NA													:=			0    		,
Standby                                             :=          1           ,
IOLP                                                :=          2           ,
PNB                                                 :=          3           ,
TBOT                                                :=          4           ,
LP_VISIONSHUTTLE_L                                  :=          1500        ,
LP_VISIONSHUTTLE_R                                  :=          1600        ,
LP_LE                                               :=          1900        ,
LP_L01                                              :=          1901        ,
LP_L02                                              :=          1902        ,
LP_RE                                               :=          1903        ,
LP_R01                                              :=          1904        ,
LP_R02                                              :=          1905        ,
LP_L                                                :=          1910        ,
LP_R                                                :=          1911        ,
LP_LE_STACKER_01                                    :=          2000        ,
LP_LE_STACKER_01_LIFT                               :=          2001        ,
LP_LE_STACKER_01_STOPPER_01                         :=          2002        ,
LP_LE_STACKER_01_STOPPER_02                         :=          2003        ,
LP_LE_STACKER_02                                    :=          2050        ,
LP_LE_STACKER_02_LIFT                               :=          2051        ,
LP_LE_STACKER_02_STOPPER_01                         :=          2052        ,
LP_LE_STACKER_02_STOPPER_02                         :=          2053        ,
LP_LE_CONVEYOR                                      :=          2200        ,
LP_LE_CONVEYOR_STACKER_01_PRE                       :=          2250        ,
LP_LE_CONVEYOR_STACKER_01                           :=          2251        ,
LP_LE_CONVEYOR_STACKER_01_POST                      :=          2252        ,
LP_LE_CONVEYOR_STACKER_02                           :=          2300        ,
LP_L01_STACKER_01                                   :=          3000        ,
LP_L01_STACKER_01_LIFT                              :=          3001        ,
LP_L01_STACKER_01_STOPPER_01                        :=          3002        ,
LP_L01_STACKER_01_STOPPER_02                        :=          3003        ,
LP_L01_STACKER_02                                   :=          3050        ,
LP_L01_STACKER_02_LIFT                              :=          3051        ,
LP_L01_STACKER_02_STOPPER_01                        :=          3052        ,
LP_L01_STACKER_02_STOPPER_02                        :=          3053        ,
LP_L01_CONVEYOR_01                                  :=          3110        ,
LP_L01_CONVEYOR_02                                  :=          3120        ,
LP_L01_CONVEYOR_STACKER_01_PRE                      :=          3125        ,
LP_L01_CONVEYOR_STACKER_01                          :=          3126        ,
LP_L01_CONVEYOR_STACKER_01_POST                     :=          3127        ,
LP_L01_CONVEYOR_STACKER_02                          :=          3128        ,
LP_L01_CONVEYOR_STACKER_02_POST                     :=          3129        ,
LP_L01_EPORT                                        :=          3130        ,
LP_L01_EPORT_STANDBY                                :=          3131        ,
LP_L01_EPORT_STOPPER_01                             :=          3132        ,
LP_L01_EPORT_STOPPER_02                             :=          3133        ,
LP_L01_VISION                                       :=          3140        ,
LP_L01_UPORT                                        :=          3151        ,
LP_L02_STACKER_01                                   :=          3200        ,
LP_L02_STACKER_01_LIFT                              :=          3201        ,
LP_L02_STACKER_01_STOPPER_01                        :=          3202        ,
LP_L02_STACKER_01_STOPPER_02                        :=          3203        ,
LP_L02_STACKER_02                                   :=          3250        ,
LP_L02_STACKER_02_LIFT                              :=          3251        ,
LP_L02_STACKER_02_STOPPER_01                        :=          3252        ,
LP_L02_STACKER_02_STOPPER_02                        :=          3253        ,
LP_L02_CONVEYOR_01                                  :=          3310        ,
LP_L02_CONVEYOR_02                                  :=          3320        ,
LP_L02_CONVEYOR_STACKER_01_PRE                      :=          3325        ,
LP_L02_CONVEYOR_STACKER_01                          :=          3326        ,
LP_L02_CONVEYOR_STACKER_01_POST                     :=          3327        ,
LP_L02_CONVEYOR_STACKER_02                          :=          3328        ,
LP_L02_CONVEYOR_STACKER_02_POST                     :=          3329        ,
LP_L02_EPORT                                        :=          3330        ,
LP_L02_EPORT_STANDBY                                :=          3331        ,
LP_L02_EPORT_STOPPER_01                             :=          3332        ,
LP_L02_EPORT_STOPPER_02                             :=          3333        ,
LP_L02_VISION                                       :=          3340        ,
LP_L02_UPORT                                        :=          3351        ,
LP_RE_STACKER_01                                    :=          4000        ,
LP_RE_STACKER_01_LIFT                               :=          4001        ,
LP_RE_STACKER_01_STOPPER_01                         :=          4002        ,
LP_RE_STACKER_01_STOPPER_02                         :=          4003        ,
LP_RE_STACKER_02                                    :=          4050        ,
LP_RE_STACKER_02_LIFT                               :=          4051        ,
LP_RE_STACKER_02_STOPPER_01                         :=          4052        ,
LP_RE_STACKER_02_STOPPER_02                         :=          4053        ,
LP_RE_CONVEYOR                                      :=          4200        ,
LP_RE_CONVEYOR_STACKER_01_PRE                       :=          4250        ,
LP_RE_CONVEYOR_STACKER_01                           :=          4251        ,
LP_RE_CONVEYOR_STACKER_01_POST                      :=          4252        ,
LP_RE_CONVEYOR_STACKER_02                           :=          4300        ,
LP_R01_STACKER_01                                   :=          5000        ,
LP_R01_STACKER_01_LIFT                              :=          5001        ,
LP_R01_STACKER_01_STOPPER_01                        :=          5002        ,
LP_R01_STACKER_01_STOPPER_02                        :=          5003        ,
LP_R01_STACKER_02                                   :=          5050        ,
LP_R01_STACKER_02_LIFT                              :=          5051        ,
LP_R01_STACKER_02_STOPPER_01                        :=          5052        ,
LP_R01_STACKER_02_STOPPER_02                        :=          5053        ,
LP_R01_CONVEYOR_01                                  :=          5110        ,
LP_R01_CONVEYOR_02                                  :=          5120        ,
LP_R01_CONVEYOR_STACKER_01_PRE                      :=          5125        ,
LP_R01_CONVEYOR_STACKER_01                          :=          5126        ,
LP_R01_CONVEYOR_STACKER_01_POST                     :=          5127        ,
LP_R01_CONVEYOR_STACKER_02                          :=          5128        ,
LP_R01_CONVEYOR_STACKER_02_POST                     :=          5129        ,
LP_R01_EPORT                                        :=          5130        ,
LP_R01_EPORT_STANDBY                                :=          5131        ,
LP_R01_EPORT_STOPPER_01                             :=          5132        ,
LP_R01_EPORT_STOPPER_02                             :=          5133        ,
LP_R01_VISION                                       :=          5140        ,
LP_R01_UPORT                                        :=          5151        ,
LP_R02_STACKER_01                                   :=          5200        ,
LP_R02_STACKER_01_LIFT                              :=          5201        ,
LP_R02_STACKER_01_STOPPER_01                        :=          5202        ,
LP_R02_STACKER_01_STOPPER_02                        :=          5203        ,
LP_R02_STACKER_02                                   :=          5250        ,
LP_R02_STACKER_02_LIFT                              :=          5251        ,
LP_R02_STACKER_02_STOPPER_01                        :=          5252        ,
LP_R02_STACKER_02_STOPPER_02                        :=          5253        ,
LP_R02_CONVEYOR_01                                  :=          5310        ,
LP_R02_CONVEYOR_02                                  :=          5320        ,
LP_R02_CONVEYOR_STACKER_01_PRE                      :=          5325        ,
LP_R02_CONVEYOR_STACKER_01                          :=          5326        ,
LP_R02_CONVEYOR_STACKER_01_POST                     :=          5327        ,
LP_R02_CONVEYOR_STACKER_02                          :=          5328        ,
LP_R02_CONVEYOR_STACKER_02_POST                     :=          5329        ,
LP_R02_EPORT                                        :=          5330        ,
LP_R02_EPORT_STANDBY                                :=          5331        ,
LP_R02_EPORT_STOPPER_01                             :=          5332        ,
LP_R02_EPORT_STOPPER_02                             :=          5333        ,
LP_R02_VISION                                       :=          5340        ,
LP_R02_UPORT                                        :=          5351        ,
TTS                                                 :=          10000       ,
TTS_SHUTTLE_01                                      :=          10100       ,
TTS_SHUTTLE_01_SERVICE                              :=          10101       ,
TTS_SHUTTLE_01_PARK                                 :=          10102       ,
TTS_SHUTTLE_01_CONVEYOR                             :=          10103       ,
TTS_SHUTTLE_02                                      :=          10200       ,
TTS_SHUTTLE_02_SERVICE                              :=          10201       ,
TTS_SHUTTLE_02_CONVEYOR                             :=          10202       ,
TTS_SHUTTLE_03                                      :=          10300       ,
TTS_SHUTTLE_03_SERVICE                              :=          10301       ,
TTS_SHUTTLE_03_PARK                                 :=          10302       ,
TTS_SHUTTLE_03_CONVEYOR                             :=          10303       ,
PNB_DOOR_TOP_LEFT                                   :=          20001       ,
PNB_DOOR_TOP_RIGHT                                  :=          20002       ,
PNB_DOOR_BOTTOM                                     :=          20003       ,
PNB_LANE_01                                         :=          21000       ,
PNB_LANE_01_CONVEYOR                                :=          21001       ,
PNB_LANE_02                                         :=          21050       ,
PNB_LANE_02_CONVEYOR                                :=          21051       ,
PNB_LANE_03                                         :=          21150       ,
PNB_LANE_03_CONVEYOR                                :=          21151       ,
PNB_LANE_04                                         :=          21200       ,
PNB_LANE_04_CONVEYOR                                :=          21201       ,
PNB_LANE_05                                         :=          21350       ,
PNB_LANE_05_CONVEYOR                                :=          21351       ,
PNB_LANE_06                                         :=          21400       ,
PNB_LANE_06_CONVEYOR                                :=          21401       ,
PNB_LANE_07                                         :=          21450       ,
PNB_LANE_07_CONVEYOR                                :=          21451       ,
PNB_LANE_08                                         :=          21500       ,
PNB_LANE_08_CONVEYOR                                :=          21501       ,
PNB_GANTRY_01                                       :=          22500       ,
PNB_GANTRY_01_PARK                                  :=          22501       ,
PNB_UPCAM_L                                         :=          22502       ,
PNB_RFID_L                                          :=          22503       ,
PNB_RFID_L_01                                       :=          22504       ,
PNB_RFID_L_02                                       :=          22505       ,
PNB_GANTRY_01_SERVICE                               :=          22506       ,
PNB_GANTRY_01_HEAD_A01                              :=          22550       ,
PNB_GANTRY_01_HEAD_A02                              :=          22560       ,
PNB_GANTRY_01_HEAD_A03                              :=          22570       ,
PNB_GANTRY_01_HEAD_A04                              :=          22580       ,
PNB_GANTRY_02                                       :=          23000       ,
PNB_GANTRY_02_PARK                                  :=          23001       ,
PNB_UPCAM_R                                         :=          23002       ,
PNB_RFID_R                                          :=          23003       ,
PNB_RFID_R_01                                       :=          23004       ,
PNB_RFID_R_02                                       :=          23005       ,
PNB_GANTRY_02_SERVICE                               :=          23006       ,
PNB_GANTRY_02_HEAD_A01                              :=          23050       ,
PNB_GANTRY_02_HEAD_A02                              :=          23060       ,
PNB_GANTRY_02_HEAD_A03                              :=          23070       ,
PNB_GANTRY_02_HEAD_A04                              :=          23080       ,
PRECISOR_UL                                         :=          24000       ,
PRECISOR_UL_CLEAN                                   :=          24001       ,
PRECISOR_UL_01                                      :=          24002       ,
PRECISOR_UL_02                                      :=          24003       ,
PRECISOR_UL_CLEAN_READID                            :=          24004       ,
PRECISOR_UL_01_READID                               :=          24005       ,
PRECISOR_UL_02_READID                               :=          24006       ,
PRECISOR_UL_A01_01                                  :=          24011       ,
PRECISOR_UL_A01_02                                  :=          24012       ,
PRECISOR_UL_A02_01                                  :=          24021       ,
PRECISOR_UL_A02_02                                  :=          24022       ,
PRECISOR_UL_A03_01                                  :=          24031       ,
PRECISOR_UL_A03_02                                  :=          24032       ,
PRECISOR_UL_A04_01                                  :=          24041       ,
PRECISOR_UL_A04_02                                  :=          24042       ,
PRECISOR_UL_B01_01                                  :=          24061       ,
PRECISOR_UL_B01_02                                  :=          24062       ,
PRECISOR_UL_B02_01                                  :=          24071       ,
PRECISOR_UL_B02_02                                  :=          24072       ,
PRECISOR_UL_B03_01                                  :=          24081       ,
PRECISOR_UL_B03_02                                  :=          24082       ,
PRECISOR_UL_B04_01                                  :=          24091       ,
PRECISOR_UL_B04_02                                  :=          24092       ,
PRECISOR_UL_C01_01                                  :=          24111       ,
PRECISOR_UL_C01_02                                  :=          24112       ,
PRECISOR_UL_C02_01                                  :=          24121       ,
PRECISOR_UL_C02_02                                  :=          24122       ,
PRECISOR_UL_C03_01                                  :=          24131       ,
PRECISOR_UL_C03_02                                  :=          24132       ,
PRECISOR_UL_C04_01                                  :=          24141       ,
PRECISOR_UL_C04_02                                  :=          24142       ,
PRECISOR_UL_D01_01                                  :=          24161       ,
PRECISOR_UL_D01_02                                  :=          24162       ,
PRECISOR_UL_D02_01                                  :=          24171       ,
PRECISOR_UL_D02_02                                  :=          24172       ,
PRECISOR_UL_D03_01                                  :=          24181       ,
PRECISOR_UL_D03_02                                  :=          24182       ,
PRECISOR_UL_D04_01                                  :=          24191       ,
PRECISOR_UL_D04_02                                  :=          24192       ,
PRECISOR_UR                                         :=          24500       ,
PRECISOR_UR_CLEAN                                   :=          24501       ,
PRECISOR_UR_01                                      :=          24502       ,
PRECISOR_UR_02                                      :=          24503       ,
PRECISOR_UR_CLEAN_READID                            :=          24504       ,
PRECISOR_UR_01_READID                               :=          24505       ,
PRECISOR_UR_02_READID                               :=          24506       ,
PRECISOR_UR_A01_01                                  :=          24511       ,
PRECISOR_UR_A01_02                                  :=          24512       ,
PRECISOR_UR_A02_01                                  :=          24521       ,
PRECISOR_UR_A02_02                                  :=          24522       ,
PRECISOR_UR_A03_01                                  :=          24531       ,
PRECISOR_UR_A03_02                                  :=          24532       ,
PRECISOR_UR_A04_01                                  :=          24541       ,
PRECISOR_UR_A04_02                                  :=          24542       ,
PRECISOR_UR_B01_01                                  :=          24561       ,
PRECISOR_UR_B01_02                                  :=          24562       ,
PRECISOR_UR_B02_01                                  :=          24571       ,
PRECISOR_UR_B02_02                                  :=          24572       ,
PRECISOR_UR_B03_01                                  :=          24581       ,
PRECISOR_UR_B03_02                                  :=          24582       ,
PRECISOR_UR_B04_01                                  :=          24591       ,
PRECISOR_UR_B04_02                                  :=          24592       ,
PRECISOR_UR_C01_01                                  :=          24611       ,
PRECISOR_UR_C01_02                                  :=          24612       ,
PRECISOR_UR_C02_01                                  :=          24621       ,
PRECISOR_UR_C02_02                                  :=          24622       ,
PRECISOR_UR_C03_01                                  :=          24631       ,
PRECISOR_UR_C03_02                                  :=          24632       ,
PRECISOR_UR_C04_01                                  :=          24641       ,
PRECISOR_UR_C04_02                                  :=          24642       ,
PRECISOR_UR_D01_01                                  :=          24661       ,
PRECISOR_UR_D01_02                                  :=          24662       ,
PRECISOR_UR_D02_01                                  :=          24671       ,
PRECISOR_UR_D02_02                                  :=          24672       ,
PRECISOR_UR_D03_01                                  :=          24681       ,
PRECISOR_UR_D03_02                                  :=          24682       ,
PRECISOR_UR_D04_01                                  :=          24691       ,
PRECISOR_UR_D04_02                                  :=          24692       ,
PRECISOR_DL                                         :=          25000       ,
PRECISOR_DL_CLEAN                                   :=          25001       ,
PRECISOR_DL_01                                      :=          25002       ,
PRECISOR_DL_02                                      :=          25003       ,
PRECISOR_DL_CLEAN_READID                            :=          25004       ,
PRECISOR_DL_01_READID                               :=          25005       ,
PRECISOR_DL_02_READID                               :=          25006       ,
PRECISOR_DL_A01_01                                  :=          25011       ,
PRECISOR_DL_A01_02                                  :=          25012       ,
PRECISOR_DL_A02_01                                  :=          25021       ,
PRECISOR_DL_A02_02                                  :=          25022       ,
PRECISOR_DL_A03_01                                  :=          25031       ,
PRECISOR_DL_A03_02                                  :=          25032       ,
PRECISOR_DL_A04_01                                  :=          25041       ,
PRECISOR_DL_A04_02                                  :=          25042       ,
PRECISOR_DL_B01_01                                  :=          25061       ,
PRECISOR_DL_B01_02                                  :=          25062       ,
PRECISOR_DL_B02_01                                  :=          25071       ,
PRECISOR_DL_B02_02                                  :=          25072       ,
PRECISOR_DL_B03_01                                  :=          25081       ,
PRECISOR_DL_B03_02                                  :=          25082       ,
PRECISOR_DL_B04_01                                  :=          25091       ,
PRECISOR_DL_B04_02                                  :=          25092       ,
PRECISOR_DL_C01_01                                  :=          25111       ,
PRECISOR_DL_C01_02                                  :=          25112       ,
PRECISOR_DL_C02_01                                  :=          25121       ,
PRECISOR_DL_C02_02                                  :=          25122       ,
PRECISOR_DL_C03_01                                  :=          25131       ,
PRECISOR_DL_C03_02                                  :=          25132       ,
PRECISOR_DL_C04_01                                  :=          25141       ,
PRECISOR_DL_C04_02                                  :=          25142       ,
PRECISOR_DL_D01_01                                  :=          25161       ,
PRECISOR_DL_D01_02                                  :=          25162       ,
PRECISOR_DL_D02_01                                  :=          25171       ,
PRECISOR_DL_D02_02                                  :=          25172       ,
PRECISOR_DL_D03_01                                  :=          25181       ,
PRECISOR_DL_D03_02                                  :=          25182       ,
PRECISOR_DL_D04_01                                  :=          25191       ,
PRECISOR_DL_D04_02                                  :=          25192       ,
PRECISOR_DR                                         :=          25500       ,
PRECISOR_DR_CLEAN                                   :=          25501       ,
PRECISOR_DR_01                                      :=          25502       ,
PRECISOR_DR_02                                      :=          25503       ,
PRECISOR_DR_CLEAN_READID                            :=          25504       ,
PRECISOR_DR_01_READID                               :=          25505       ,
PRECISOR_DR_02_READID                               :=          25506       ,
PRECISOR_DR_A01_01                                  :=          25511       ,
PRECISOR_DR_A01_02                                  :=          25512       ,
PRECISOR_DR_A02_01                                  :=          25521       ,
PRECISOR_DR_A02_02                                  :=          25522       ,
PRECISOR_DR_A03_01                                  :=          25531       ,
PRECISOR_DR_A03_02                                  :=          25532       ,
PRECISOR_DR_A04_01                                  :=          25541       ,
PRECISOR_DR_A04_02                                  :=          25542       ,
PRECISOR_DR_B01_01                                  :=          25561       ,
PRECISOR_DR_B01_02                                  :=          25562       ,
PRECISOR_DR_B02_01                                  :=          25571       ,
PRECISOR_DR_B02_02                                  :=          25572       ,
PRECISOR_DR_B03_01                                  :=          25581       ,
PRECISOR_DR_B03_02                                  :=          25582       ,
PRECISOR_DR_B04_01                                  :=          25591       ,
PRECISOR_DR_B04_02                                  :=          25592       ,
PRECISOR_DR_C01_01                                  :=          25611       ,
PRECISOR_DR_C01_02                                  :=          25612       ,
PRECISOR_DR_C02_01                                  :=          25621       ,
PRECISOR_DR_C02_02                                  :=          25622       ,
PRECISOR_DR_C03_01                                  :=          25631       ,
PRECISOR_DR_C03_02                                  :=          25632       ,
PRECISOR_DR_C04_01                                  :=          25641       ,
PRECISOR_DR_C04_02                                  :=          25642       ,
PRECISOR_DR_D01_01                                  :=          25661       ,
PRECISOR_DR_D01_02                                  :=          25662       ,
PRECISOR_DR_D02_01                                  :=          25671       ,
PRECISOR_DR_D02_02                                  :=          25672       ,
PRECISOR_DR_D03_01                                  :=          25681       ,
PRECISOR_DR_D03_02                                  :=          25682       ,
PRECISOR_DR_D04_01                                  :=          25691       ,
PRECISOR_DR_D04_02                                  :=          25692       ,
TBOT_L                                              :=          30000       ,
TBOT_L_RFID                                         :=          30001       ,
TBOT_L_SERVICE                                      :=          30002       ,
TBOT_L_PARK                                         :=          30003       ,
TBOT_L_HEAD_A01                                     :=          30020       ,
TBOT_L_HEAD_A02                                     :=          30040       ,
TBOT_L_HEAD_A03                                     :=          30060       ,
TBOT_L_HEAD_A04                                     :=          30080       ,
TBOT_L_HEAD_B01                                     :=          30100       ,
TBOT_L_HEAD_B02                                     :=          30120       ,
TBOT_L_HEAD_B03                                     :=          30140       ,
TBOT_L_HEAD_B04                                     :=          30160       ,
TBOT_L_HEAD_C01                                     :=          30180       ,
TBOT_L_HEAD_C02                                     :=          30200       ,
TBOT_L_HEAD_C03                                     :=          30220       ,
TBOT_L_HEAD_C04                                     :=          30240       ,
TBOT_L_HEAD_D01                                     :=          30260       ,
TBOT_L_HEAD_D02                                     :=          30280       ,
TBOT_L_HEAD_D03                                     :=          30300       ,
TBOT_L_HEAD_D04                                     :=          30320       ,
TBOT_R                                              :=          30500       ,
TBOT_R_RFID                                         :=          30501       ,
TBOT_R_SERVICE                                      :=          30502       ,
TBOT_R_PARK                                         :=          30503       ,
TBOT_R_HEAD_A01                                     :=          30520       ,
TBOT_R_HEAD_A02                                     :=          30540       ,
TBOT_R_HEAD_A03                                     :=          30560       ,
TBOT_R_HEAD_A04                                     :=          30580       ,
TBOT_R_HEAD_B01                                     :=          30600       ,
TBOT_R_HEAD_B02                                     :=          30620       ,
TBOT_R_HEAD_B03                                     :=          30640       ,
TBOT_R_HEAD_B04                                     :=          30660       ,
TBOT_R_HEAD_C01                                     :=          30680       ,
TBOT_R_HEAD_C02                                     :=          30700       ,
TBOT_R_HEAD_C03                                     :=          30720       ,
TBOT_R_HEAD_C04                                     :=          30740       ,
TBOT_R_HEAD_D01                                     :=          30760       ,
TBOT_R_HEAD_D02                                     :=          30780       ,
TBOT_R_HEAD_D03                                     :=          30800       ,
TBOT_R_HEAD_D04                                     :=          30820       ,
COLUMN_LA                                           :=          35000       ,
COLUMN_LB                                           :=          35100       ,
COLUMN_LC                                           :=          35200       ,
COLUMN_RA                                           :=          35300       ,
COLUMN_RB                                           :=          35400       ,
COLUMN_RC                                           :=          35500       ,
LEVEL_LA01                                          :=          36000       ,
LEVEL_LA02                                          :=          36010       ,
LEVEL_LA03                                          :=          36020       ,
LEVEL_LA04                                          :=          36030       ,
LEVEL_LA05                                          :=          36040       ,
LEVEL_LA06                                          :=          36050       ,
LEVEL_LB01                                          :=          36060       ,
LEVEL_LB02                                          :=          36070       ,
LEVEL_LB03                                          :=          36080       ,
LEVEL_LB04                                          :=          36090       ,
LEVEL_LB05                                          :=          36100       ,
LEVEL_LB06                                          :=          36110       ,
LEVEL_LC01                                          :=          36120       ,
LEVEL_LC02                                          :=          36130       ,
LEVEL_LC03                                          :=          36140       ,
LEVEL_LC04                                          :=          36150       ,
LEVEL_LC05                                          :=          36160       ,
LEVEL_LC06                                          :=          36170       ,
LEVEL_RA01                                          :=          37000       ,
LEVEL_RA02                                          :=          37010       ,
LEVEL_RA03                                          :=          37020       ,
LEVEL_RA04                                          :=          37030       ,
LEVEL_RA05                                          :=          37040       ,
LEVEL_RA06                                          :=          37050       ,
LEVEL_RB01                                          :=          37060       ,
LEVEL_RB02                                          :=          37070       ,
LEVEL_RB03                                          :=          37080       ,
LEVEL_RB04                                          :=          37090       ,
LEVEL_RB05                                          :=          37100       ,
LEVEL_RB06                                          :=          37110       ,
LEVEL_RC01                                          :=          37120       ,
LEVEL_RC02                                          :=          37130       ,
LEVEL_RC03                                          :=          37140       ,
LEVEL_RC04                                          :=          37150       ,
LEVEL_RC05                                          :=          37160       ,
LEVEL_RC06                                          :=          37170       ,
CELL_LA101_TESTER                                   :=          45000       ,
CELL_LA101_TESTER_SOCKET_A01                        :=          45001       ,
CELL_LA101_TESTER_SOCKET_A02                        :=          45002       ,
CELL_LA101_TESTER_SOCKET_A03                        :=          45003       ,
CELL_LA101_TESTER_SOCKET_A04                        :=          45004       ,
CELL_LA101_TESTER_SOCKET_B01                        :=          45011       ,
CELL_LA101_TESTER_SOCKET_B02                        :=          45012       ,
CELL_LA101_TESTER_SOCKET_B03                        :=          45013       ,
CELL_LA101_TESTER_SOCKET_B04                        :=          45014       ,
CELL_LA101_TESTER_SOCKET_C01                        :=          45021       ,
CELL_LA101_TESTER_SOCKET_C02                        :=          45022       ,
CELL_LA101_TESTER_SOCKET_C03                        :=          45023       ,
CELL_LA101_TESTER_SOCKET_C04                        :=          45024       ,
CELL_LA101_TESTER_SOCKET_D01                        :=          45031       ,
CELL_LA101_TESTER_SOCKET_D02                        :=          45032       ,
CELL_LA101_TESTER_SOCKET_D03                        :=          45033       ,
CELL_LA101_TESTER_SOCKET_D04                        :=          45034       ,
CELL_LA101_TESTER_FRONT                             :=          45035       ,
CELL_LA101_AP                                       :=          45050       ,
CELL_LA101_AP_TH_A01                                :=          45051       ,
CELL_LA101_AP_TH_A02                                :=          45052       ,
CELL_LA101_AP_TH_A03                                :=          45053       ,
CELL_LA101_AP_TH_A04                                :=          45054       ,
CELL_LA101_AP_TH_B01                                :=          45061       ,
CELL_LA101_AP_TH_B02                                :=          45062       ,
CELL_LA101_AP_TH_B03                                :=          45063       ,
CELL_LA101_AP_TH_B04                                :=          45064       ,
CELL_LA101_AP_TH_C01                                :=          45071       ,
CELL_LA101_AP_TH_C02                                :=          45072       ,
CELL_LA101_AP_TH_C03                                :=          45073       ,
CELL_LA101_AP_TH_C04                                :=          45074       ,
CELL_LA101_AP_TH_D01                                :=          45081       ,
CELL_LA101_AP_TH_D02                                :=          45082       ,
CELL_LA101_AP_TH_D03                                :=          45083       ,
CELL_LA101_AP_TH_D04                                :=          45084       ,
CELL_LA201_TESTER                                   :=          45100       ,
CELL_LA201_TESTER_SOCKET_A01                        :=          45101       ,
CELL_LA201_TESTER_SOCKET_A02                        :=          45102       ,
CELL_LA201_TESTER_SOCKET_A03                        :=          45103       ,
CELL_LA201_TESTER_SOCKET_A04                        :=          45104       ,
CELL_LA201_TESTER_SOCKET_B01                        :=          45111       ,
CELL_LA201_TESTER_SOCKET_B02                        :=          45112       ,
CELL_LA201_TESTER_SOCKET_B03                        :=          45113       ,
CELL_LA201_TESTER_SOCKET_B04                        :=          45114       ,
CELL_LA201_TESTER_SOCKET_C01                        :=          45121       ,
CELL_LA201_TESTER_SOCKET_C02                        :=          45122       ,
CELL_LA201_TESTER_SOCKET_C03                        :=          45123       ,
CELL_LA201_TESTER_SOCKET_C04                        :=          45124       ,
CELL_LA201_TESTER_SOCKET_D01                        :=          45131       ,
CELL_LA201_TESTER_SOCKET_D02                        :=          45132       ,
CELL_LA201_TESTER_SOCKET_D03                        :=          45133       ,
CELL_LA201_TESTER_SOCKET_D04                        :=          45134       ,
CELL_LA201_TESTER_FRONT                             :=          45135       ,
CELL_LA201_AP                                       :=          45150       ,
CELL_LA201_AP_TH_A01                                :=          45151       ,
CELL_LA201_AP_TH_A02                                :=          45152       ,
CELL_LA201_AP_TH_A03                                :=          45153       ,
CELL_LA201_AP_TH_A04                                :=          45154       ,
CELL_LA201_AP_TH_B01                                :=          45161       ,
CELL_LA201_AP_TH_B02                                :=          45162       ,
CELL_LA201_AP_TH_B03                                :=          45163       ,
CELL_LA201_AP_TH_B04                                :=          45164       ,
CELL_LA201_AP_TH_C01                                :=          45171       ,
CELL_LA201_AP_TH_C02                                :=          45172       ,
CELL_LA201_AP_TH_C03                                :=          45173       ,
CELL_LA201_AP_TH_C04                                :=          45174       ,
CELL_LA201_AP_TH_D01                                :=          45181       ,
CELL_LA201_AP_TH_D02                                :=          45182       ,
CELL_LA201_AP_TH_D03                                :=          45183       ,
CELL_LA201_AP_TH_D04                                :=          45184       ,
CELL_LA301_TESTER                                   :=          45200       ,
CELL_LA301_TESTER_SOCKET_A01                        :=          45201       ,
CELL_LA301_TESTER_SOCKET_A02                        :=          45202       ,
CELL_LA301_TESTER_SOCKET_A03                        :=          45203       ,
CELL_LA301_TESTER_SOCKET_A04                        :=          45204       ,
CELL_LA301_TESTER_SOCKET_B01                        :=          45211       ,
CELL_LA301_TESTER_SOCKET_B02                        :=          45212       ,
CELL_LA301_TESTER_SOCKET_B03                        :=          45213       ,
CELL_LA301_TESTER_SOCKET_B04                        :=          45214       ,
CELL_LA301_TESTER_SOCKET_C01                        :=          45221       ,
CELL_LA301_TESTER_SOCKET_C02                        :=          45222       ,
CELL_LA301_TESTER_SOCKET_C03                        :=          45223       ,
CELL_LA301_TESTER_SOCKET_C04                        :=          45224       ,
CELL_LA301_TESTER_SOCKET_D01                        :=          45231       ,
CELL_LA301_TESTER_SOCKET_D02                        :=          45232       ,
CELL_LA301_TESTER_SOCKET_D03                        :=          45233       ,
CELL_LA301_TESTER_SOCKET_D04                        :=          45234       ,
CELL_LA301_AP                                       :=          45250       ,
CELL_LA301_AP_TH_A01                                :=          45251       ,
CELL_LA301_AP_TH_A02                                :=          45252       ,
CELL_LA301_AP_TH_A03                                :=          45253       ,
CELL_LA301_AP_TH_A04                                :=          45254       ,
CELL_LA301_AP_TH_B01                                :=          45261       ,
CELL_LA301_AP_TH_B02                                :=          45262       ,
CELL_LA301_AP_TH_B03                                :=          45263       ,
CELL_LA301_AP_TH_B04                                :=          45264       ,
CELL_LA301_AP_TH_C01                                :=          45271       ,
CELL_LA301_AP_TH_C02                                :=          45272       ,
CELL_LA301_AP_TH_C03                                :=          45273       ,
CELL_LA301_AP_TH_C04                                :=          45274       ,
CELL_LA301_AP_TH_D01                                :=          45281       ,
CELL_LA301_AP_TH_D02                                :=          45282       ,
CELL_LA301_AP_TH_D03                                :=          45283       ,
CELL_LA301_AP_TH_D04                                :=          45284       ,
CELL_LA401_TESTER                                   :=          45300       ,
CELL_LA401_TESTER_SOCKET_A01                        :=          45301       ,
CELL_LA401_TESTER_SOCKET_A02                        :=          45302       ,
CELL_LA401_TESTER_SOCKET_A03                        :=          45303       ,
CELL_LA401_TESTER_SOCKET_A04                        :=          45304       ,
CELL_LA401_TESTER_SOCKET_B01                        :=          45311       ,
CELL_LA401_TESTER_SOCKET_B02                        :=          45312       ,
CELL_LA401_TESTER_SOCKET_B03                        :=          45313       ,
CELL_LA401_TESTER_SOCKET_B04                        :=          45314       ,
CELL_LA401_TESTER_SOCKET_C01                        :=          45321       ,
CELL_LA401_TESTER_SOCKET_C02                        :=          45322       ,
CELL_LA401_TESTER_SOCKET_C03                        :=          45323       ,
CELL_LA401_TESTER_SOCKET_C04                        :=          45324       ,
CELL_LA401_TESTER_SOCKET_D01                        :=          45331       ,
CELL_LA401_TESTER_SOCKET_D02                        :=          45332       ,
CELL_LA401_TESTER_SOCKET_D03                        :=          45333       ,
CELL_LA401_TESTER_SOCKET_D04                        :=          45334       ,
CELL_LA401_AP                                       :=          45350       ,
CELL_LA401_AP_TH_A01                                :=          45351       ,
CELL_LA401_AP_TH_A02                                :=          45352       ,
CELL_LA401_AP_TH_A03                                :=          45353       ,
CELL_LA401_AP_TH_A04                                :=          45354       ,
CELL_LA401_AP_TH_B01                                :=          45361       ,
CELL_LA401_AP_TH_B02                                :=          45362       ,
CELL_LA401_AP_TH_B03                                :=          45363       ,
CELL_LA401_AP_TH_B04                                :=          45364       ,
CELL_LA401_AP_TH_C01                                :=          45371       ,
CELL_LA401_AP_TH_C02                                :=          45372       ,
CELL_LA401_AP_TH_C03                                :=          45373       ,
CELL_LA401_AP_TH_C04                                :=          45374       ,
CELL_LA401_AP_TH_D01                                :=          45381       ,
CELL_LA401_AP_TH_D02                                :=          45382       ,
CELL_LA401_AP_TH_D03                                :=          45383       ,
CELL_LA401_AP_TH_D04                                :=          45384       ,
CELL_LA501_TESTER                                   :=          45400       ,
CELL_LA501_TESTER_SOCKET_A01                        :=          45401       ,
CELL_LA501_TESTER_SOCKET_A02                        :=          45402       ,
CELL_LA501_TESTER_SOCKET_A03                        :=          45403       ,
CELL_LA501_TESTER_SOCKET_A04                        :=          45404       ,
CELL_LA501_TESTER_SOCKET_B01                        :=          45411       ,
CELL_LA501_TESTER_SOCKET_B02                        :=          45412       ,
CELL_LA501_TESTER_SOCKET_B03                        :=          45413       ,
CELL_LA501_TESTER_SOCKET_B04                        :=          45414       ,
CELL_LA501_TESTER_SOCKET_C01                        :=          45421       ,
CELL_LA501_TESTER_SOCKET_C02                        :=          45422       ,
CELL_LA501_TESTER_SOCKET_C03                        :=          45423       ,
CELL_LA501_TESTER_SOCKET_C04                        :=          45424       ,
CELL_LA501_TESTER_SOCKET_D01                        :=          45431       ,
CELL_LA501_TESTER_SOCKET_D02                        :=          45432       ,
CELL_LA501_TESTER_SOCKET_D03                        :=          45433       ,
CELL_LA501_TESTER_SOCKET_D04                        :=          45434       ,
CELL_LA501_AP                                       :=          45450       ,
CELL_LA501_AP_TH_A01                                :=          45451       ,
CELL_LA501_AP_TH_A02                                :=          45452       ,
CELL_LA501_AP_TH_A03                                :=          45453       ,
CELL_LA501_AP_TH_A04                                :=          45454       ,
CELL_LA501_AP_TH_B01                                :=          45461       ,
CELL_LA501_AP_TH_B02                                :=          45462       ,
CELL_LA501_AP_TH_B03                                :=          45463       ,
CELL_LA501_AP_TH_B04                                :=          45464       ,
CELL_LA501_AP_TH_C01                                :=          45471       ,
CELL_LA501_AP_TH_C02                                :=          45472       ,
CELL_LA501_AP_TH_C03                                :=          45473       ,
CELL_LA501_AP_TH_C04                                :=          45474       ,
CELL_LA501_AP_TH_D01                                :=          45481       ,
CELL_LA501_AP_TH_D02                                :=          45482       ,
CELL_LA501_AP_TH_D03                                :=          45483       ,
CELL_LA501_AP_TH_D04                                :=          45484       ,
CELL_LA601_TESTER                                   :=          45500       ,
CELL_LA601_TESTER_SOCKET_A01                        :=          45501       ,
CELL_LA601_TESTER_SOCKET_A02                        :=          45502       ,
CELL_LA601_TESTER_SOCKET_A03                        :=          45503       ,
CELL_LA601_TESTER_SOCKET_A04                        :=          45504       ,
CELL_LA601_TESTER_SOCKET_B01                        :=          45511       ,
CELL_LA601_TESTER_SOCKET_B02                        :=          45512       ,
CELL_LA601_TESTER_SOCKET_B03                        :=          45513       ,
CELL_LA601_TESTER_SOCKET_B04                        :=          45514       ,
CELL_LA601_TESTER_SOCKET_C01                        :=          45521       ,
CELL_LA601_TESTER_SOCKET_C02                        :=          45522       ,
CELL_LA601_TESTER_SOCKET_C03                        :=          45523       ,
CELL_LA601_TESTER_SOCKET_C04                        :=          45524       ,
CELL_LA601_TESTER_SOCKET_D01                        :=          45531       ,
CELL_LA601_TESTER_SOCKET_D02                        :=          45532       ,
CELL_LA601_TESTER_SOCKET_D03                        :=          45533       ,
CELL_LA601_TESTER_SOCKET_D04                        :=          45534       ,
CELL_LA601_AP                                       :=          45550       ,
CELL_LA601_AP_TH_A01                                :=          45551       ,
CELL_LA601_AP_TH_A02                                :=          45552       ,
CELL_LA601_AP_TH_A03                                :=          45553       ,
CELL_LA601_AP_TH_A04                                :=          45554       ,
CELL_LA601_AP_TH_B01                                :=          45561       ,
CELL_LA601_AP_TH_B02                                :=          45562       ,
CELL_LA601_AP_TH_B03                                :=          45563       ,
CELL_LA601_AP_TH_B04                                :=          45564       ,
CELL_LA601_AP_TH_C01                                :=          45571       ,
CELL_LA601_AP_TH_C02                                :=          45572       ,
CELL_LA601_AP_TH_C03                                :=          45573       ,
CELL_LA601_AP_TH_C04                                :=          45574       ,
CELL_LA601_AP_TH_D01                                :=          45581       ,
CELL_LA601_AP_TH_D02                                :=          45582       ,
CELL_LA601_AP_TH_D03                                :=          45583       ,
CELL_LA601_AP_TH_D04                                :=          45584       ,
CELL_LB101_TESTER                                   :=          46000       ,
CELL_LB101_TESTER_SOCKET_A01                        :=          46001       ,
CELL_LB101_TESTER_SOCKET_A02                        :=          46002       ,
CELL_LB101_TESTER_SOCKET_A03                        :=          46003       ,
CELL_LB101_TESTER_SOCKET_A04                        :=          46004       ,
CELL_LB101_TESTER_SOCKET_B01                        :=          46011       ,
CELL_LB101_TESTER_SOCKET_B02                        :=          46012       ,
CELL_LB101_TESTER_SOCKET_B03                        :=          46013       ,
CELL_LB101_TESTER_SOCKET_B04                        :=          46014       ,
CELL_LB101_TESTER_SOCKET_C01                        :=          46021       ,
CELL_LB101_TESTER_SOCKET_C02                        :=          46022       ,
CELL_LB101_TESTER_SOCKET_C03                        :=          46023       ,
CELL_LB101_TESTER_SOCKET_C04                        :=          46024       ,
CELL_LB101_TESTER_SOCKET_D01                        :=          46031       ,
CELL_LB101_TESTER_SOCKET_D02                        :=          46032       ,
CELL_LB101_TESTER_SOCKET_D03                        :=          46033       ,
CELL_LB101_TESTER_SOCKET_D04                        :=          46034       ,
CELL_LB101_AP                                       :=          46050       ,
CELL_LB101_AP_TH_A01                                :=          46051       ,
CELL_LB101_AP_TH_A02                                :=          46052       ,
CELL_LB101_AP_TH_A03                                :=          46053       ,
CELL_LB101_AP_TH_A04                                :=          46054       ,
CELL_LB101_AP_TH_B01                                :=          46061       ,
CELL_LB101_AP_TH_B02                                :=          46062       ,
CELL_LB101_AP_TH_B03                                :=          46063       ,
CELL_LB101_AP_TH_B04                                :=          46064       ,
CELL_LB101_AP_TH_C01                                :=          46071       ,
CELL_LB101_AP_TH_C02                                :=          46072       ,
CELL_LB101_AP_TH_C03                                :=          46073       ,
CELL_LB101_AP_TH_C04                                :=          46074       ,
CELL_LB101_AP_TH_D01                                :=          46081       ,
CELL_LB101_AP_TH_D02                                :=          46082       ,
CELL_LB101_AP_TH_D03                                :=          46083       ,
CELL_LB101_AP_TH_D04                                :=          46084       ,
CELL_LB201_TESTER                                   :=          46100       ,
CELL_LB201_TESTER_SOCKET_A01                        :=          46101       ,
CELL_LB201_TESTER_SOCKET_A02                        :=          46102       ,
CELL_LB201_TESTER_SOCKET_A03                        :=          46103       ,
CELL_LB201_TESTER_SOCKET_A04                        :=          46104       ,
CELL_LB201_TESTER_SOCKET_B01                        :=          46111       ,
CELL_LB201_TESTER_SOCKET_B02                        :=          46112       ,
CELL_LB201_TESTER_SOCKET_B03                        :=          46113       ,
CELL_LB201_TESTER_SOCKET_B04                        :=          46114       ,
CELL_LB201_TESTER_SOCKET_C01                        :=          46121       ,
CELL_LB201_TESTER_SOCKET_C02                        :=          46122       ,
CELL_LB201_TESTER_SOCKET_C03                        :=          46123       ,
CELL_LB201_TESTER_SOCKET_C04                        :=          46124       ,
CELL_LB201_TESTER_SOCKET_D01                        :=          46131       ,
CELL_LB201_TESTER_SOCKET_D02                        :=          46132       ,
CELL_LB201_TESTER_SOCKET_D03                        :=          46133       ,
CELL_LB201_TESTER_SOCKET_D04                        :=          46134       ,
CELL_LB201_AP                                       :=          46150       ,
CELL_LB201_AP_TH_A01                                :=          46151       ,
CELL_LB201_AP_TH_A02                                :=          46152       ,
CELL_LB201_AP_TH_A03                                :=          46153       ,
CELL_LB201_AP_TH_A04                                :=          46154       ,
CELL_LB201_AP_TH_B01                                :=          46161       ,
CELL_LB201_AP_TH_B02                                :=          46162       ,
CELL_LB201_AP_TH_B03                                :=          46163       ,
CELL_LB201_AP_TH_B04                                :=          46164       ,
CELL_LB201_AP_TH_C01                                :=          46171       ,
CELL_LB201_AP_TH_C02                                :=          46172       ,
CELL_LB201_AP_TH_C03                                :=          46173       ,
CELL_LB201_AP_TH_C04                                :=          46174       ,
CELL_LB201_AP_TH_D01                                :=          46181       ,
CELL_LB201_AP_TH_D02                                :=          46182       ,
CELL_LB201_AP_TH_D03                                :=          46183       ,
CELL_LB201_AP_TH_D04                                :=          46184       ,
CELL_LB301_TESTER                                   :=          46200       ,
CELL_LB301_TESTER_SOCKET_A01                        :=          46201       ,
CELL_LB301_TESTER_SOCKET_A02                        :=          46202       ,
CELL_LB301_TESTER_SOCKET_A03                        :=          46203       ,
CELL_LB301_TESTER_SOCKET_A04                        :=          46204       ,
CELL_LB301_TESTER_SOCKET_B01                        :=          46211       ,
CELL_LB301_TESTER_SOCKET_B02                        :=          46212       ,
CELL_LB301_TESTER_SOCKET_B03                        :=          46213       ,
CELL_LB301_TESTER_SOCKET_B04                        :=          46214       ,
CELL_LB301_TESTER_SOCKET_C01                        :=          46221       ,
CELL_LB301_TESTER_SOCKET_C02                        :=          46222       ,
CELL_LB301_TESTER_SOCKET_C03                        :=          46223       ,
CELL_LB301_TESTER_SOCKET_C04                        :=          46224       ,
CELL_LB301_TESTER_SOCKET_D01                        :=          46231       ,
CELL_LB301_TESTER_SOCKET_D02                        :=          46232       ,
CELL_LB301_TESTER_SOCKET_D03                        :=          46233       ,
CELL_LB301_TESTER_SOCKET_D04                        :=          46234       ,
CELL_LB301_AP                                       :=          46250       ,
CELL_LB301_AP_TH_A01                                :=          46251       ,
CELL_LB301_AP_TH_A02                                :=          46252       ,
CELL_LB301_AP_TH_A03                                :=          46253       ,
CELL_LB301_AP_TH_A04                                :=          46254       ,
CELL_LB301_AP_TH_B01                                :=          46261       ,
CELL_LB301_AP_TH_B02                                :=          46262       ,
CELL_LB301_AP_TH_B03                                :=          46263       ,
CELL_LB301_AP_TH_B04                                :=          46264       ,
CELL_LB301_AP_TH_C01                                :=          46271       ,
CELL_LB301_AP_TH_C02                                :=          46272       ,
CELL_LB301_AP_TH_C03                                :=          46273       ,
CELL_LB301_AP_TH_C04                                :=          46274       ,
CELL_LB301_AP_TH_D01                                :=          46281       ,
CELL_LB301_AP_TH_D02                                :=          46282       ,
CELL_LB301_AP_TH_D03                                :=          46283       ,
CELL_LB301_AP_TH_D04                                :=          46284       ,
CELL_LB401_TESTER                                   :=          46300       ,
CELL_LB401_TESTER_SOCKET_A01                        :=          46301       ,
CELL_LB401_TESTER_SOCKET_A02                        :=          46302       ,
CELL_LB401_TESTER_SOCKET_A03                        :=          46303       ,
CELL_LB401_TESTER_SOCKET_A04                        :=          46304       ,
CELL_LB401_TESTER_SOCKET_B01                        :=          46311       ,
CELL_LB401_TESTER_SOCKET_B02                        :=          46312       ,
CELL_LB401_TESTER_SOCKET_B03                        :=          46313       ,
CELL_LB401_TESTER_SOCKET_B04                        :=          46314       ,
CELL_LB401_TESTER_SOCKET_C01                        :=          46321       ,
CELL_LB401_TESTER_SOCKET_C02                        :=          46322       ,
CELL_LB401_TESTER_SOCKET_C03                        :=          46323       ,
CELL_LB401_TESTER_SOCKET_C04                        :=          46324       ,
CELL_LB401_TESTER_SOCKET_D01                        :=          46331       ,
CELL_LB401_TESTER_SOCKET_D02                        :=          46332       ,
CELL_LB401_TESTER_SOCKET_D03                        :=          46333       ,
CELL_LB401_TESTER_SOCKET_D04                        :=          46334       ,
CELL_LB401_AP                                       :=          46350       ,
CELL_LB401_AP_TH_A01                                :=          46351       ,
CELL_LB401_AP_TH_A02                                :=          46352       ,
CELL_LB401_AP_TH_A03                                :=          46353       ,
CELL_LB401_AP_TH_A04                                :=          46354       ,
CELL_LB401_AP_TH_B01                                :=          46361       ,
CELL_LB401_AP_TH_B02                                :=          46362       ,
CELL_LB401_AP_TH_B03                                :=          46363       ,
CELL_LB401_AP_TH_B04                                :=          46364       ,
CELL_LB401_AP_TH_C01                                :=          46371       ,
CELL_LB401_AP_TH_C02                                :=          46372       ,
CELL_LB401_AP_TH_C03                                :=          46373       ,
CELL_LB401_AP_TH_C04                                :=          46374       ,
CELL_LB401_AP_TH_D01                                :=          46381       ,
CELL_LB401_AP_TH_D02                                :=          46382       ,
CELL_LB401_AP_TH_D03                                :=          46383       ,
CELL_LB401_AP_TH_D04                                :=          46384       ,
CELL_LB501_TESTER                                   :=          46400       ,
CELL_LB501_TESTER_SOCKET_A01                        :=          46401       ,
CELL_LB501_TESTER_SOCKET_A02                        :=          46402       ,
CELL_LB501_TESTER_SOCKET_A03                        :=          46403       ,
CELL_LB501_TESTER_SOCKET_A04                        :=          46404       ,
CELL_LB501_TESTER_SOCKET_B01                        :=          46411       ,
CELL_LB501_TESTER_SOCKET_B02                        :=          46412       ,
CELL_LB501_TESTER_SOCKET_B03                        :=          46413       ,
CELL_LB501_TESTER_SOCKET_B04                        :=          46414       ,
CELL_LB501_TESTER_SOCKET_C01                        :=          46421       ,
CELL_LB501_TESTER_SOCKET_C02                        :=          46422       ,
CELL_LB501_TESTER_SOCKET_C03                        :=          46423       ,
CELL_LB501_TESTER_SOCKET_C04                        :=          46424       ,
CELL_LB501_TESTER_SOCKET_D01                        :=          46431       ,
CELL_LB501_TESTER_SOCKET_D02                        :=          46432       ,
CELL_LB501_TESTER_SOCKET_D03                        :=          46433       ,
CELL_LB501_TESTER_SOCKET_D04                        :=          46434       ,
CELL_LB501_AP                                       :=          46450       ,
CELL_LB501_AP_TH_A01                                :=          46451       ,
CELL_LB501_AP_TH_A02                                :=          46452       ,
CELL_LB501_AP_TH_A03                                :=          46453       ,
CELL_LB501_AP_TH_A04                                :=          46454       ,
CELL_LB501_AP_TH_B01                                :=          46461       ,
CELL_LB501_AP_TH_B02                                :=          46462       ,
CELL_LB501_AP_TH_B03                                :=          46463       ,
CELL_LB501_AP_TH_B04                                :=          46464       ,
CELL_LB501_AP_TH_C01                                :=          46471       ,
CELL_LB501_AP_TH_C02                                :=          46472       ,
CELL_LB501_AP_TH_C03                                :=          46473       ,
CELL_LB501_AP_TH_C04                                :=          46474       ,
CELL_LB501_AP_TH_D01                                :=          46481       ,
CELL_LB501_AP_TH_D02                                :=          46482       ,
CELL_LB501_AP_TH_D03                                :=          46483       ,
CELL_LB501_AP_TH_D04                                :=          46484       ,
CELL_LB601_TESTER                                   :=          46500       ,
CELL_LB601_TESTER_SOCKET_A01                        :=          46501       ,
CELL_LB601_TESTER_SOCKET_A02                        :=          46502       ,
CELL_LB601_TESTER_SOCKET_A03                        :=          46503       ,
CELL_LB601_TESTER_SOCKET_A04                        :=          46504       ,
CELL_LB601_TESTER_SOCKET_B01                        :=          46511       ,
CELL_LB601_TESTER_SOCKET_B02                        :=          46512       ,
CELL_LB601_TESTER_SOCKET_B03                        :=          46513       ,
CELL_LB601_TESTER_SOCKET_B04                        :=          46514       ,
CELL_LB601_TESTER_SOCKET_C01                        :=          46521       ,
CELL_LB601_TESTER_SOCKET_C02                        :=          46522       ,
CELL_LB601_TESTER_SOCKET_C03                        :=          46523       ,
CELL_LB601_TESTER_SOCKET_C04                        :=          46524       ,
CELL_LB601_TESTER_SOCKET_D01                        :=          46531       ,
CELL_LB601_TESTER_SOCKET_D02                        :=          46532       ,
CELL_LB601_TESTER_SOCKET_D03                        :=          46533       ,
CELL_LB601_TESTER_SOCKET_D04                        :=          46534       ,
CELL_LB601_AP                                       :=          46550       ,
CELL_LB601_AP_TH_A01                                :=          46551       ,
CELL_LB601_AP_TH_A02                                :=          46552       ,
CELL_LB601_AP_TH_A03                                :=          46553       ,
CELL_LB601_AP_TH_A04                                :=          46554       ,
CELL_LB601_AP_TH_B01                                :=          46561       ,
CELL_LB601_AP_TH_B02                                :=          46562       ,
CELL_LB601_AP_TH_B03                                :=          46563       ,
CELL_LB601_AP_TH_B04                                :=          46564       ,
CELL_LB601_AP_TH_C01                                :=          46571       ,
CELL_LB601_AP_TH_C02                                :=          46572       ,
CELL_LB601_AP_TH_C03                                :=          46573       ,
CELL_LB601_AP_TH_C04                                :=          46574       ,
CELL_LB601_AP_TH_D01                                :=          46581       ,
CELL_LB601_AP_TH_D02                                :=          46582       ,
CELL_LB601_AP_TH_D03                                :=          46583       ,
CELL_LB601_AP_TH_D04                                :=          46584       ,
CELL_LC101_TESTER                                   :=          47000       ,
CELL_LC101_TESTER_SOCKET_A01                        :=          47001       ,
CELL_LC101_TESTER_SOCKET_A02                        :=          47002       ,
CELL_LC101_TESTER_SOCKET_A03                        :=          47003       ,
CELL_LC101_TESTER_SOCKET_A04                        :=          47004       ,
CELL_LC101_TESTER_SOCKET_B01                        :=          47011       ,
CELL_LC101_TESTER_SOCKET_B02                        :=          47012       ,
CELL_LC101_TESTER_SOCKET_B03                        :=          47013       ,
CELL_LC101_TESTER_SOCKET_B04                        :=          47014       ,
CELL_LC101_TESTER_SOCKET_C01                        :=          47021       ,
CELL_LC101_TESTER_SOCKET_C02                        :=          47022       ,
CELL_LC101_TESTER_SOCKET_C03                        :=          47023       ,
CELL_LC101_TESTER_SOCKET_C04                        :=          47024       ,
CELL_LC101_TESTER_SOCKET_D01                        :=          47031       ,
CELL_LC101_TESTER_SOCKET_D02                        :=          47032       ,
CELL_LC101_TESTER_SOCKET_D03                        :=          47033       ,
CELL_LC101_TESTER_SOCKET_D04                        :=          47034       ,
CELL_LC101_AP                                       :=          47050       ,
CELL_LC101_AP_TH_A01                                :=          47051       ,
CELL_LC101_AP_TH_A02                                :=          47052       ,
CELL_LC101_AP_TH_A03                                :=          47053       ,
CELL_LC101_AP_TH_A04                                :=          47054       ,
CELL_LC101_AP_TH_B01                                :=          47061       ,
CELL_LC101_AP_TH_B02                                :=          47062       ,
CELL_LC101_AP_TH_B03                                :=          47063       ,
CELL_LC101_AP_TH_B04                                :=          47064       ,
CELL_LC101_AP_TH_C01                                :=          47071       ,
CELL_LC101_AP_TH_C02                                :=          47072       ,
CELL_LC101_AP_TH_C03                                :=          47073       ,
CELL_LC101_AP_TH_C04                                :=          47074       ,
CELL_LC101_AP_TH_D01                                :=          47081       ,
CELL_LC101_AP_TH_D02                                :=          47082       ,
CELL_LC101_AP_TH_D03                                :=          47083       ,
CELL_LC101_AP_TH_D04                                :=          47084       ,
CELL_LC201_TESTER                                   :=          47100       ,
CELL_LC201_TESTER_SOCKET_A01                        :=          47101       ,
CELL_LC201_TESTER_SOCKET_A02                        :=          47102       ,
CELL_LC201_TESTER_SOCKET_A03                        :=          47103       ,
CELL_LC201_TESTER_SOCKET_A04                        :=          47104       ,
CELL_LC201_TESTER_SOCKET_B01                        :=          47111       ,
CELL_LC201_TESTER_SOCKET_B02                        :=          47112       ,
CELL_LC201_TESTER_SOCKET_B03                        :=          47113       ,
CELL_LC201_TESTER_SOCKET_B04                        :=          47114       ,
CELL_LC201_TESTER_SOCKET_C01                        :=          47121       ,
CELL_LC201_TESTER_SOCKET_C02                        :=          47122       ,
CELL_LC201_TESTER_SOCKET_C03                        :=          47123       ,
CELL_LC201_TESTER_SOCKET_C04                        :=          47124       ,
CELL_LC201_TESTER_SOCKET_D01                        :=          47131       ,
CELL_LC201_TESTER_SOCKET_D02                        :=          47132       ,
CELL_LC201_TESTER_SOCKET_D03                        :=          47133       ,
CELL_LC201_TESTER_SOCKET_D04                        :=          47134       ,
CELL_LC201_AP                                       :=          47150       ,
CELL_LC201_AP_TH_A01                                :=          47151       ,
CELL_LC201_AP_TH_A02                                :=          47152       ,
CELL_LC201_AP_TH_A03                                :=          47153       ,
CELL_LC201_AP_TH_A04                                :=          47154       ,
CELL_LC201_AP_TH_B01                                :=          47161       ,
CELL_LC201_AP_TH_B02                                :=          47162       ,
CELL_LC201_AP_TH_B03                                :=          47163       ,
CELL_LC201_AP_TH_B04                                :=          47164       ,
CELL_LC201_AP_TH_C01                                :=          47171       ,
CELL_LC201_AP_TH_C02                                :=          47172       ,
CELL_LC201_AP_TH_C03                                :=          47173       ,
CELL_LC201_AP_TH_C04                                :=          47174       ,
CELL_LC201_AP_TH_D01                                :=          47181       ,
CELL_LC201_AP_TH_D02                                :=          47182       ,
CELL_LC201_AP_TH_D03                                :=          47183       ,
CELL_LC201_AP_TH_D04                                :=          47184       ,
CELL_LC301_TESTER                                   :=          47200       ,
CELL_LC301_TESTER_SOCKET_A01                        :=          47201       ,
CELL_LC301_TESTER_SOCKET_A02                        :=          47202       ,
CELL_LC301_TESTER_SOCKET_A03                        :=          47203       ,
CELL_LC301_TESTER_SOCKET_A04                        :=          47204       ,
CELL_LC301_TESTER_SOCKET_B01                        :=          47211       ,
CELL_LC301_TESTER_SOCKET_B02                        :=          47212       ,
CELL_LC301_TESTER_SOCKET_B03                        :=          47213       ,
CELL_LC301_TESTER_SOCKET_B04                        :=          47214       ,
CELL_LC301_TESTER_SOCKET_C01                        :=          47221       ,
CELL_LC301_TESTER_SOCKET_C02                        :=          47222       ,
CELL_LC301_TESTER_SOCKET_C03                        :=          47223       ,
CELL_LC301_TESTER_SOCKET_C04                        :=          47224       ,
CELL_LC301_TESTER_SOCKET_D01                        :=          47231       ,
CELL_LC301_TESTER_SOCKET_D02                        :=          47232       ,
CELL_LC301_TESTER_SOCKET_D03                        :=          47233       ,
CELL_LC301_TESTER_SOCKET_D04                        :=          47234       ,
CELL_LC301_AP                                       :=          47250       ,
CELL_LC301_AP_TH_A01                                :=          47251       ,
CELL_LC301_AP_TH_A02                                :=          47252       ,
CELL_LC301_AP_TH_A03                                :=          47253       ,
CELL_LC301_AP_TH_A04                                :=          47254       ,
CELL_LC301_AP_TH_B01                                :=          47261       ,
CELL_LC301_AP_TH_B02                                :=          47262       ,
CELL_LC301_AP_TH_B03                                :=          47263       ,
CELL_LC301_AP_TH_B04                                :=          47264       ,
CELL_LC301_AP_TH_C01                                :=          47271       ,
CELL_LC301_AP_TH_C02                                :=          47272       ,
CELL_LC301_AP_TH_C03                                :=          47273       ,
CELL_LC301_AP_TH_C04                                :=          47274       ,
CELL_LC301_AP_TH_D01                                :=          47281       ,
CELL_LC301_AP_TH_D02                                :=          47282       ,
CELL_LC301_AP_TH_D03                                :=          47283       ,
CELL_LC301_AP_TH_D04                                :=          47284       ,
CELL_LC401_TESTER                                   :=          47300       ,
CELL_LC401_TESTER_SOCKET_A01                        :=          47301       ,
CELL_LC401_TESTER_SOCKET_A02                        :=          47302       ,
CELL_LC401_TESTER_SOCKET_A03                        :=          47303       ,
CELL_LC401_TESTER_SOCKET_A04                        :=          47304       ,
CELL_LC401_TESTER_SOCKET_B01                        :=          47311       ,
CELL_LC401_TESTER_SOCKET_B02                        :=          47312       ,
CELL_LC401_TESTER_SOCKET_B03                        :=          47313       ,
CELL_LC401_TESTER_SOCKET_B04                        :=          47314       ,
CELL_LC401_TESTER_SOCKET_C01                        :=          47321       ,
CELL_LC401_TESTER_SOCKET_C02                        :=          47322       ,
CELL_LC401_TESTER_SOCKET_C03                        :=          47323       ,
CELL_LC401_TESTER_SOCKET_C04                        :=          47324       ,
CELL_LC401_TESTER_SOCKET_D01                        :=          47331       ,
CELL_LC401_TESTER_SOCKET_D02                        :=          47332       ,
CELL_LC401_TESTER_SOCKET_D03                        :=          47333       ,
CELL_LC401_TESTER_SOCKET_D04                        :=          47334       ,
CELL_LC401_AP                                       :=          47350       ,
CELL_LC401_AP_TH_A01                                :=          47351       ,
CELL_LC401_AP_TH_A02                                :=          47352       ,
CELL_LC401_AP_TH_A03                                :=          47353       ,
CELL_LC401_AP_TH_A04                                :=          47354       ,
CELL_LC401_AP_TH_B01                                :=          47361       ,
CELL_LC401_AP_TH_B02                                :=          47362       ,
CELL_LC401_AP_TH_B03                                :=          47363       ,
CELL_LC401_AP_TH_B04                                :=          47364       ,
CELL_LC401_AP_TH_C01                                :=          47371       ,
CELL_LC401_AP_TH_C02                                :=          47372       ,
CELL_LC401_AP_TH_C03                                :=          47373       ,
CELL_LC401_AP_TH_C04                                :=          47374       ,
CELL_LC401_AP_TH_D01                                :=          47381       ,
CELL_LC401_AP_TH_D02                                :=          47382       ,
CELL_LC401_AP_TH_D03                                :=          47383       ,
CELL_LC401_AP_TH_D04                                :=          47384       ,
CELL_LC501_TESTER                                   :=          47400       ,
CELL_LC501_TESTER_SOCKET_A01                        :=          47401       ,
CELL_LC501_TESTER_SOCKET_A02                        :=          47402       ,
CELL_LC501_TESTER_SOCKET_A03                        :=          47403       ,
CELL_LC501_TESTER_SOCKET_A04                        :=          47404       ,
CELL_LC501_TESTER_SOCKET_B01                        :=          47411       ,
CELL_LC501_TESTER_SOCKET_B02                        :=          47412       ,
CELL_LC501_TESTER_SOCKET_B03                        :=          47413       ,
CELL_LC501_TESTER_SOCKET_B04                        :=          47414       ,
CELL_LC501_TESTER_SOCKET_C01                        :=          47421       ,
CELL_LC501_TESTER_SOCKET_C02                        :=          47422       ,
CELL_LC501_TESTER_SOCKET_C03                        :=          47423       ,
CELL_LC501_TESTER_SOCKET_C04                        :=          47424       ,
CELL_LC501_TESTER_SOCKET_D01                        :=          47431       ,
CELL_LC501_TESTER_SOCKET_D02                        :=          47432       ,
CELL_LC501_TESTER_SOCKET_D03                        :=          47433       ,
CELL_LC501_TESTER_SOCKET_D04                        :=          47434       ,
CELL_LC501_AP                                       :=          47450       ,
CELL_LC501_AP_TH_A01                                :=          47451       ,
CELL_LC501_AP_TH_A02                                :=          47452       ,
CELL_LC501_AP_TH_A03                                :=          47453       ,
CELL_LC501_AP_TH_A04                                :=          47454       ,
CELL_LC501_AP_TH_B01                                :=          47461       ,
CELL_LC501_AP_TH_B02                                :=          47462       ,
CELL_LC501_AP_TH_B03                                :=          47463       ,
CELL_LC501_AP_TH_B04                                :=          47464       ,
CELL_LC501_AP_TH_C01                                :=          47471       ,
CELL_LC501_AP_TH_C02                                :=          47472       ,
CELL_LC501_AP_TH_C03                                :=          47473       ,
CELL_LC501_AP_TH_C04                                :=          47474       ,
CELL_LC501_AP_TH_D01                                :=          47481       ,
CELL_LC501_AP_TH_D02                                :=          47482       ,
CELL_LC501_AP_TH_D03                                :=          47483       ,
CELL_LC501_AP_TH_D04                                :=          47484       ,
CELL_LC601_TESTER                                   :=          47500       ,
CELL_LC601_TESTER_SOCKET_A01                        :=          47501       ,
CELL_LC601_TESTER_SOCKET_A02                        :=          47502       ,
CELL_LC601_TESTER_SOCKET_A03                        :=          47503       ,
CELL_LC601_TESTER_SOCKET_A04                        :=          47504       ,
CELL_LC601_TESTER_SOCKET_B01                        :=          47511       ,
CELL_LC601_TESTER_SOCKET_B02                        :=          47512       ,
CELL_LC601_TESTER_SOCKET_B03                        :=          47513       ,
CELL_LC601_TESTER_SOCKET_B04                        :=          47514       ,
CELL_LC601_TESTER_SOCKET_C01                        :=          47521       ,
CELL_LC601_TESTER_SOCKET_C02                        :=          47522       ,
CELL_LC601_TESTER_SOCKET_C03                        :=          47523       ,
CELL_LC601_TESTER_SOCKET_C04                        :=          47524       ,
CELL_LC601_TESTER_SOCKET_D01                        :=          47531       ,
CELL_LC601_TESTER_SOCKET_D02                        :=          47532       ,
CELL_LC601_TESTER_SOCKET_D03                        :=          47533       ,
CELL_LC601_TESTER_SOCKET_D04                        :=          47534       ,
CELL_LC601_AP                                       :=          47550       ,
CELL_LC601_AP_TH_A01                                :=          47551       ,
CELL_LC601_AP_TH_A02                                :=          47552       ,
CELL_LC601_AP_TH_A03                                :=          47553       ,
CELL_LC601_AP_TH_A04                                :=          47554       ,
CELL_LC601_AP_TH_B01                                :=          47561       ,
CELL_LC601_AP_TH_B02                                :=          47562       ,
CELL_LC601_AP_TH_B03                                :=          47563       ,
CELL_LC601_AP_TH_B04                                :=          47564       ,
CELL_LC601_AP_TH_C01                                :=          47571       ,
CELL_LC601_AP_TH_C02                                :=          47572       ,
CELL_LC601_AP_TH_C03                                :=          47573       ,
CELL_LC601_AP_TH_C04                                :=          47574       ,
CELL_LC601_AP_TH_D01                                :=          47581       ,
CELL_LC601_AP_TH_D02                                :=          47582       ,
CELL_LC601_AP_TH_D03                                :=          47583       ,
CELL_LC601_AP_TH_D04                                :=          47584       ,
CELL_RA101_TESTER                                   :=          50000       ,
CELL_RA101_TESTER_SOCKET_A01                        :=          50001       ,
CELL_RA101_TESTER_SOCKET_A02                        :=          50002       ,
CELL_RA101_TESTER_SOCKET_A03                        :=          50003       ,
CELL_RA101_TESTER_SOCKET_A04                        :=          50004       ,
CELL_RA101_TESTER_SOCKET_B01                        :=          50011       ,
CELL_RA101_TESTER_SOCKET_B02                        :=          50012       ,
CELL_RA101_TESTER_SOCKET_B03                        :=          50013       ,
CELL_RA101_TESTER_SOCKET_B04                        :=          50014       ,
CELL_RA101_TESTER_SOCKET_C01                        :=          50021       ,
CELL_RA101_TESTER_SOCKET_C02                        :=          50022       ,
CELL_RA101_TESTER_SOCKET_C03                        :=          50023       ,
CELL_RA101_TESTER_SOCKET_C04                        :=          50024       ,
CELL_RA101_TESTER_SOCKET_D01                        :=          50031       ,
CELL_RA101_TESTER_SOCKET_D02                        :=          50032       ,
CELL_RA101_TESTER_SOCKET_D03                        :=          50033       ,
CELL_RA101_TESTER_SOCKET_D04                        :=          50034       ,
CELL_RA101_AP                                       :=          50050       ,
CELL_RA101_AP_TH_A01                                :=          50051       ,
CELL_RA101_AP_TH_A02								:=          50052       ,
CELL_RA101_AP_TH_A03                                :=          50053       ,
CELL_RA101_AP_TH_A04                                :=          50054       ,
CELL_RA101_AP_TH_B01                                :=          50061       ,
CELL_RA101_AP_TH_B02                                :=          50062       ,
CELL_RA101_AP_TH_B03                                :=          50063       ,
CELL_RA101_AP_TH_B04                                :=          50064       ,
CELL_RA101_AP_TH_C01                                :=          50071       ,
CELL_RA101_AP_TH_C02                                :=          50072       ,
CELL_RA101_AP_TH_C03                                :=          50073       ,
CELL_RA101_AP_TH_C04                                :=          50074       ,
CELL_RA101_AP_TH_D01                                :=          50081       ,
CELL_RA101_AP_TH_D02                                :=          50082       ,
CELL_RA101_AP_TH_D03                                :=          50083       ,
CELL_RA101_AP_TH_D04                                :=          50084       ,
CELL_RA201_TESTER                                   :=          50100       ,
CELL_RA201_TESTER_SOCKET_A01                        :=          50101       ,
CELL_RA201_TESTER_SOCKET_A02                        :=          50102       ,
CELL_RA201_TESTER_SOCKET_A03                        :=          50103       ,
CELL_RA201_TESTER_SOCKET_A04                        :=          50104       ,
CELL_RA201_TESTER_SOCKET_B01                        :=          50111       ,
CELL_RA201_TESTER_SOCKET_B02                        :=          50112       ,
CELL_RA201_TESTER_SOCKET_B03                        :=          50113       ,
CELL_RA201_TESTER_SOCKET_B04                        :=          50114       ,
CELL_RA201_TESTER_SOCKET_C01                        :=          50121       ,
CELL_RA201_TESTER_SOCKET_C02                        :=          50122       ,
CELL_RA201_TESTER_SOCKET_C03                        :=          50123       ,
CELL_RA201_TESTER_SOCKET_C04                        :=          50124       ,
CELL_RA201_TESTER_SOCKET_D01                        :=          50131       ,
CELL_RA201_TESTER_SOCKET_D02                        :=          50132       ,
CELL_RA201_TESTER_SOCKET_D03                        :=          50133       ,
CELL_RA201_TESTER_SOCKET_D04                        :=          50134       ,
CELL_RA201_AP                                       :=          50150       ,
CELL_RA201_AP_TH_A01                                :=          50151       ,
CELL_RA201_AP_TH_A02                                :=          50152       ,
CELL_RA201_AP_TH_A03                                :=          50153       ,
CELL_RA201_AP_TH_A04                                :=          50154       ,
CELL_RA201_AP_TH_B01                                :=          50161       ,
CELL_RA201_AP_TH_B02                                :=          50162       ,
CELL_RA201_AP_TH_B03                                :=          50163       ,
CELL_RA201_AP_TH_B04                                :=          50164       ,
CELL_RA201_AP_TH_C01                                :=          50171       ,
CELL_RA201_AP_TH_C02                                :=          50172       ,
CELL_RA201_AP_TH_C03                                :=          50173       ,
CELL_RA201_AP_TH_C04                                :=          50174       ,
CELL_RA201_AP_TH_D01                                :=          50181       ,
CELL_RA201_AP_TH_D02                                :=          50182       ,
CELL_RA201_AP_TH_D03                                :=          50183       ,
CELL_RA201_AP_TH_D04                                :=          50184       ,
CELL_RA301_TESTER                                   :=          50200       ,
CELL_RA301_TESTER_SOCKET_A01                        :=          50201       ,
CELL_RA301_TESTER_SOCKET_A02                        :=          50202       ,
CELL_RA301_TESTER_SOCKET_A03                        :=          50203       ,
CELL_RA301_TESTER_SOCKET_A04                        :=          50204       ,
CELL_RA301_TESTER_SOCKET_B01                        :=          50211       ,
CELL_RA301_TESTER_SOCKET_B02                        :=          50212       ,
CELL_RA301_TESTER_SOCKET_B03                        :=          50213       ,
CELL_RA301_TESTER_SOCKET_B04                        :=          50214       ,
CELL_RA301_TESTER_SOCKET_C01                        :=          50221       ,
CELL_RA301_TESTER_SOCKET_C02                        :=          50222       ,
CELL_RA301_TESTER_SOCKET_C03                        :=          50223       ,
CELL_RA301_TESTER_SOCKET_C04                        :=          50224       ,
CELL_RA301_TESTER_SOCKET_D01                        :=          50231       ,
CELL_RA301_TESTER_SOCKET_D02                        :=          50232       ,
CELL_RA301_TESTER_SOCKET_D03                        :=          50233       ,
CELL_RA301_TESTER_SOCKET_D04                        :=          50234       ,
CELL_RA301_AP                                       :=          50250       ,
CELL_RA301_AP_TH_A01                                :=          50251       ,
CELL_RA301_AP_TH_A02                                :=          50252       ,
CELL_RA301_AP_TH_A03                                :=          50253       ,
CELL_RA301_AP_TH_A04                                :=          50254       ,
CELL_RA301_AP_TH_B01                                :=          50261       ,
CELL_RA301_AP_TH_B02                                :=          50262       ,
CELL_RA301_AP_TH_B03                                :=          50263       ,
CELL_RA301_AP_TH_B04                                :=          50264       ,
CELL_RA301_AP_TH_C01                                :=          50271       ,
CELL_RA301_AP_TH_C02                                :=          50272       ,
CELL_RA301_AP_TH_C03                                :=          50273       ,
CELL_RA301_AP_TH_C04                                :=          50274       ,
CELL_RA301_AP_TH_D01                                :=          50281       ,
CELL_RA301_AP_TH_D02                                :=          50282       ,
CELL_RA301_AP_TH_D03                                :=          50283       ,
CELL_RA301_AP_TH_D04                                :=          50284       ,
CELL_RA401_TESTER                                   :=          50300       ,
CELL_RA401_TESTER_SOCKET_A01                        :=          50301       ,
CELL_RA401_TESTER_SOCKET_A02                        :=          50302       ,
CELL_RA401_TESTER_SOCKET_A03                        :=          50303       ,
CELL_RA401_TESTER_SOCKET_A04                        :=          50304       ,
CELL_RA401_TESTER_SOCKET_B01                        :=          50311       ,
CELL_RA401_TESTER_SOCKET_B02                        :=          50312       ,
CELL_RA401_TESTER_SOCKET_B03                        :=          50313       ,
CELL_RA401_TESTER_SOCKET_B04                        :=          50314       ,
CELL_RA401_TESTER_SOCKET_C01                        :=          50321       ,
CELL_RA401_TESTER_SOCKET_C02                        :=          50322       ,
CELL_RA401_TESTER_SOCKET_C03                        :=          50323       ,
CELL_RA401_TESTER_SOCKET_C04                        :=          50324       ,
CELL_RA401_TESTER_SOCKET_D01                        :=          50331       ,
CELL_RA401_TESTER_SOCKET_D02                        :=          50332       ,
CELL_RA401_TESTER_SOCKET_D03                        :=          50333       ,
CELL_RA401_TESTER_SOCKET_D04                        :=          50334       ,
CELL_RA401_AP                                       :=          50350       ,
CELL_RA401_AP_TH_A01                                :=          50351       ,
CELL_RA401_AP_TH_A02                                :=          50352       ,
CELL_RA401_AP_TH_A03                                :=          50353       ,
CELL_RA401_AP_TH_A04                                :=          50354       ,
CELL_RA401_AP_TH_B01                                :=          50361       ,
CELL_RA401_AP_TH_B02                                :=          50362       ,
CELL_RA401_AP_TH_B03                                :=          50363       ,
CELL_RA401_AP_TH_B04                                :=          50364       ,
CELL_RA401_AP_TH_C01                                :=          50371       ,
CELL_RA401_AP_TH_C02                                :=          50372       ,
CELL_RA401_AP_TH_C03                                :=          50373       ,
CELL_RA401_AP_TH_C04                                :=          50374       ,
CELL_RA401_AP_TH_D01                                :=          50381       ,
CELL_RA401_AP_TH_D02                                :=          50382       ,
CELL_RA401_AP_TH_D03                                :=          50383       ,
CELL_RA401_AP_TH_D04                                :=          50384       ,
CELL_RA501_TESTER                                   :=          50400       ,
CELL_RA501_TESTER_SOCKET_A01                        :=          50401       ,
CELL_RA501_TESTER_SOCKET_A02                        :=          50402       ,
CELL_RA501_TESTER_SOCKET_A03                        :=          50403       ,
CELL_RA501_TESTER_SOCKET_A04                        :=          50404       ,
CELL_RA501_TESTER_SOCKET_B01                        :=          50411       ,
CELL_RA501_TESTER_SOCKET_B02                        :=          50412       ,
CELL_RA501_TESTER_SOCKET_B03                        :=          50413       ,
CELL_RA501_TESTER_SOCKET_B04                        :=          50414       ,
CELL_RA501_TESTER_SOCKET_C01                        :=          50421       ,
CELL_RA501_TESTER_SOCKET_C02                        :=          50422       ,
CELL_RA501_TESTER_SOCKET_C03                        :=          50423       ,
CELL_RA501_TESTER_SOCKET_C04                        :=          50424       ,
CELL_RA501_TESTER_SOCKET_D01                        :=          50431       ,
CELL_RA501_TESTER_SOCKET_D02                        :=          50432       ,
CELL_RA501_TESTER_SOCKET_D03                        :=          50433       ,
CELL_RA501_TESTER_SOCKET_D04                        :=          50434       ,
CELL_RA501_AP                                       :=          50450       ,
CELL_RA501_AP_TH_A01                                :=          50451       ,
CELL_RA501_AP_TH_A02                                :=          50452       ,
CELL_RA501_AP_TH_A03                                :=          50453       ,
CELL_RA501_AP_TH_A04                                :=          50454       ,
CELL_RA501_AP_TH_B01                                :=          50461       ,
CELL_RA501_AP_TH_B02                                :=          50462       ,
CELL_RA501_AP_TH_B03                                :=          50463       ,
CELL_RA501_AP_TH_B04                                :=          50464       ,
CELL_RA501_AP_TH_C01                                :=          50471       ,
CELL_RA501_AP_TH_C02                                :=          50472       ,
CELL_RA501_AP_TH_C03                                :=          50473       ,
CELL_RA501_AP_TH_C04                                :=          50474       ,
CELL_RA501_AP_TH_D01                                :=          50481       ,
CELL_RA501_AP_TH_D02                                :=          50482       ,
CELL_RA501_AP_TH_D03                                :=          50483       ,
CELL_RA501_AP_TH_D04                                :=          50484       ,
CELL_RA601_TESTER                                   :=          50500       ,
CELL_RA601_TESTER_SOCKET_A01                        :=          50501       ,
CELL_RA601_TESTER_SOCKET_A02                        :=          50502       ,
CELL_RA601_TESTER_SOCKET_A03                        :=          50503       ,
CELL_RA601_TESTER_SOCKET_A04                        :=          50504       ,
CELL_RA601_TESTER_SOCKET_B01                        :=          50511       ,
CELL_RA601_TESTER_SOCKET_B02                        :=          50512       ,
CELL_RA601_TESTER_SOCKET_B03                        :=          50513       ,
CELL_RA601_TESTER_SOCKET_B04                        :=          50514       ,
CELL_RA601_TESTER_SOCKET_C01                        :=          50521       ,
CELL_RA601_TESTER_SOCKET_C02                        :=          50522       ,
CELL_RA601_TESTER_SOCKET_C03                        :=          50523       ,
CELL_RA601_TESTER_SOCKET_C04                        :=          50524       ,
CELL_RA601_TESTER_SOCKET_D01                        :=          50531       ,
CELL_RA601_TESTER_SOCKET_D02                        :=          50532       ,
CELL_RA601_TESTER_SOCKET_D03                        :=          50533       ,
CELL_RA601_TESTER_SOCKET_D04                        :=          50534       ,
CELL_RA601_AP                                       :=          50550       ,
CELL_RA601_AP_TH_A01                                :=          50551       ,
CELL_RA601_AP_TH_A02                                :=          50552       ,
CELL_RA601_AP_TH_A03                                :=          50553       ,
CELL_RA601_AP_TH_A04                                :=          50554       ,
CELL_RA601_AP_TH_B01                                :=          50561       ,
CELL_RA601_AP_TH_B02                                :=          50562       ,
CELL_RA601_AP_TH_B03                                :=          50563       ,
CELL_RA601_AP_TH_B04                                :=          50564       ,
CELL_RA601_AP_TH_C01                                :=          50571       ,
CELL_RA601_AP_TH_C02                                :=          50572       ,
CELL_RA601_AP_TH_C03                                :=          50573       ,
CELL_RA601_AP_TH_C04                                :=          50574       ,
CELL_RA601_AP_TH_D01                                :=          50581       ,
CELL_RA601_AP_TH_D02                                :=          50582       ,
CELL_RA601_AP_TH_D03                                :=          50583       ,
CELL_RA601_AP_TH_D04                                :=          50584       ,
CELL_RB101_TESTER                                   :=          51000       ,
CELL_RB101_TESTER_SOCKET_A01                        :=          51001       ,
CELL_RB101_TESTER_SOCKET_A02                        :=          51002       ,
CELL_RB101_TESTER_SOCKET_A03                        :=          51003       ,
CELL_RB101_TESTER_SOCKET_A04                        :=          51004       ,
CELL_RB101_TESTER_SOCKET_B01                        :=          51011       ,
CELL_RB101_TESTER_SOCKET_B02                        :=          51012       ,
CELL_RB101_TESTER_SOCKET_B03                        :=          51013       ,
CELL_RB101_TESTER_SOCKET_B04                        :=          51014       ,
CELL_RB101_TESTER_SOCKET_C01                        :=          51021       ,
CELL_RB101_TESTER_SOCKET_C02                        :=          51022       ,
CELL_RB101_TESTER_SOCKET_C03                        :=          51023       ,
CELL_RB101_TESTER_SOCKET_C04                        :=          51024       ,
CELL_RB101_TESTER_SOCKET_D01                        :=          51031       ,
CELL_RB101_TESTER_SOCKET_D02                        :=          51032       ,
CELL_RB101_TESTER_SOCKET_D03                        :=          51033       ,
CELL_RB101_TESTER_SOCKET_D04                        :=          51034       ,
CELL_RB101_AP                                       :=          51050       ,
CELL_RB101_AP_TH_A01                                :=          51051       ,
CELL_RB101_AP_TH_A02                                :=          51052       ,
CELL_RB101_AP_TH_A03                                :=          51053       ,
CELL_RB101_AP_TH_A04                                :=          51054       ,
CELL_RB101_AP_TH_B01                                :=          51061       ,
CELL_RB101_AP_TH_B02                                :=          51062       ,
CELL_RB101_AP_TH_B03                                :=          51063       ,
CELL_RB101_AP_TH_B04                                :=          51064       ,
CELL_RB101_AP_TH_C01                                :=          51071       ,
CELL_RB101_AP_TH_C02                                :=          51072       ,
CELL_RB101_AP_TH_C03                                :=          51073       ,
CELL_RB101_AP_TH_C04                                :=          51074       ,
CELL_RB101_AP_TH_D01                                :=          51081       ,
CELL_RB101_AP_TH_D02                                :=          51082       ,
CELL_RB101_AP_TH_D03                                :=          51083       ,
CELL_RB101_AP_TH_D04                                :=          51084       ,
CELL_RB201_TESTER                                   :=          51100       ,
CELL_RB201_TESTER_SOCKET_A01                        :=          51101       ,
CELL_RB201_TESTER_SOCKET_A02                        :=          51102       ,
CELL_RB201_TESTER_SOCKET_A03                        :=          51103       ,
CELL_RB201_TESTER_SOCKET_A04                        :=          51104       ,
CELL_RB201_TESTER_SOCKET_B01                        :=          51111       ,
CELL_RB201_TESTER_SOCKET_B02                        :=          51112       ,
CELL_RB201_TESTER_SOCKET_B03                        :=          51113       ,
CELL_RB201_TESTER_SOCKET_B04                        :=          51114       ,
CELL_RB201_TESTER_SOCKET_C01                        :=          51121       ,
CELL_RB201_TESTER_SOCKET_C02                        :=          51122       ,
CELL_RB201_TESTER_SOCKET_C03                        :=          51123       ,
CELL_RB201_TESTER_SOCKET_C04                        :=          51124       ,
CELL_RB201_TESTER_SOCKET_D01                        :=          51131       ,
